// TIA Portal V19 export
TYPE "C701_VAR_KMI_TYPIC"
   STRUCT
      BST { ExternalAccessible := 'False'; ExternalVisible := 'False'; ExternalWritable := 'False'} : USInt;   // Bestuurbaarheid
   END_STRUCT;
END_TYPE
